// Hata kodları için ENUM
TYPE E_CompensationError :
(
    ERROR_NONE := 0,                        // Hata yok
    ERROR_INVALID_GROUP_COUNT := 1,         // Geçersiz grup sayısı
    ERROR_NEGATIVE_POWER := 2,              // Negatif güç değeri
    ERROR_NEGATIVE_QUANTITY := 3,           // Negatif kondansatör sayısı
    ERROR_MAX_CAPACITOR_EXCEEDED := 4      // Maksimum kondansatör sayısı aşıldı
);
END_TYPE

(* stored: Version 1.1.0.1, ProductVersion 3.1.4024.15
   EnumerationTextList E_CompensationError: Id {8f7b59d6-fb11-4564-bac7-2bdab9a8b9ea} *)
